TYPE (* IEC61131-3, Table 14#5 *)
  (* Standard: 1131-3 *)
  (* Version 0.0, 1/8/2024, Cheyan, Schneider Electric, Template *)
  PACKAGE Main;
  {SET_ATTRIBUTE(nxtDataType, JT5dSobJiODsYuYBrz+XyKAFGuO9uJQ3CbgfKu/xKW+6m95wBMd6VUbwToVoS8iyuNRqTOmtzaT3TUCa1XwKFOJStHQCV/FQBSHSmPvJ+6kvpSFOGf63LdZn3qKyjU3+GSMGtmwYiPA=)}
  ACT : STRUCT
    general : BOOL;
    q : Quality;
    t : TimeStamp;
  END_STRUCT;
END_TYPE
